# EPICS substitutions: opcpaepsApp/Db/eps_temp_monitor.substitutions
file eps_temp_monitor.template {
  pattern
    {ID}
    {"01"}
    {"02"}
    {"03"}
    {"04"}
    {"05"}
    {"06"}
    {"07"}
    {"08"}
}
